FUNCTION_BLOCK PressureSensor IMPLEMENTS ITF_AnalogSensor
VAR_INPUT
END_VAR
VAR_OUTPUT
END_VAR
VAR
	//Hardware
	AI_CurrentPressure AT %I* : INT;
END_VAR

PROPERTY Value : INT
GET
Value := AI_CurrentPressure;
END_GET
END_PROPERTY

END_FUNCTION_BLOCK

(* stored: Version 1.1.0.1
   POU PressureSensor: Id {59f41b0c-fe3f-4a18-8102-d8a9230f1f3e}, SpecialFunc None
   Property Value: Id {76923876-d0ff-433e-ba41-3b8128a5ff54}
   Get Get: Id {7bd872fc-f399-4e8d-a6dd-2286fcc33c96} *)
